// TwinCAT 3 PLC project TPA
// ProgramVersion: 3.1.4023.0
// libraries:
//   Tc2_MC2, * (Beckhoff Automation GmbH)
//   Tc2_Standard, * (Beckhoff Automation GmbH)
//   Tc2_System, * (Beckhoff Automation GmbH)
//   Tc2_Utilities, * (Beckhoff Automation GmbH)
//   Tc3_Module, * (Beckhoff Automation GmbH)
//   VisuSymbols,3.5.10.0,System
// project tree:
//   / GlobalTextList.TcGTLO, PlcTask.TcTTO, Visualization Manager.TcVMO (not stored)
//   GVLs/ GVL.TcGVL
//   POUs/ MAIN.TcPOU, PlixHandler.TcPOU, POU.TcPOU
//   VISUs/ Visualization.TcVIS
// real-time tasks:
//   TASK PlcTask: cycle T#10ms, priority 20, ADS port 350
// motion (NC):
//   TASK NC-Task 1 SAF: cycle T#2ms, priority 4, ADS port 501
//   TASK NC-Task 1 SVB: cycle T#10ms, priority 8, ADS port 511
//   AXIS Axis 1 (id 1)
//     Dynamic: Acceleration=7555.57, Deceleration=7555.57, Jerk=32111.1
//     PositionAreaControl: Range=10
//     TargetPosControl: Range=10, Time=0.05
//     OtherSettings: AllowMotionCmdToSlave=true
//     encoder EncType=4
//       EncPara: ScaleFactorNumerator=0.09, MaxCount=#x0000ffff
//         Inc: RefSoftSyncMask=#x0000ffff
//     drive DrvType=24
//       Analog: VeloReferenz=1800, TorqueSetpointScale=10, ScaleFactorActTorque=0.1
//       TimeComp: TaskDelayCycles=1
//     controller CtrType=1
//       CtrPara: PriorControlFactor=1
//         PosDiffControl: Enable=false
//         Observer: BandWidth=20
// I/O:
//   DEVICE Device 3 (EtherCAT), AmsNetId 192.168.1.97.4.1
//     Box 2 (EasyCAT 32+32 rev 1) [Generic 32+32 bytes rev 1]
//     Term 3 (EK1100) [EK1100 EtherCAT Coupler (2A E-Bus)]
//       Term 4 (EL7041) [EL7041 1Ch. Stepper motor output stage (50V, 5A)]
//       Term 5 (EL9011) [EL9011 End Terminal]
// variable links:
//   NC-Task 1 SAF/Axes/Axis 1 <-> Device 3 (EtherCAT)/Term 3 (EK1100)/Term 4 (EL7041)
//     Drive/Inputs/In/nState1 @bit 3 <-> STM Status/Status/Error
//     Drive/Inputs/In/nState1 @bit 5 <-> STM Status/Status/Moving negative
//     Drive/Inputs/In/nState1 @bit 4 <-> STM Status/Status/Moving positive
//     Drive/Inputs/In/nState1 @bit 1 <-> STM Status/Status/Ready
//     Drive/Inputs/In/nState1 <-> STM Status/Status/Ready to enable
//     Drive/Inputs/In/nState1 @bit 6 <-> STM Status/Status/Torque reduced
//     Drive/Inputs/In/nState1 @bit 2 <-> STM Status/Status/Warning
//     Drive/Inputs/In/nState2 @bit 3 <-> STM Status/Status/Digital input 1
//     Drive/Inputs/In/nState2 @bit 4 <-> STM Status/Status/Digital input 2
//     Drive/Inputs/In/nState2 @bit 5 <-> STM Status/Status/Sync error
//     Drive/Inputs/In/nState2 @bit 7 <-> STM Status/Status/TxPDO Toggle
//     Drive/Inputs/In/nState4 @bit 1 <-> WcState/InputToggle
//     Drive/Inputs/In/nState4 <-> WcState/WcState
//     Drive/Outputs/Out/nCtrl1 <-> STM Control/Control/Enable
//     Drive/Outputs/Out/nCtrl1 @bit 2 <-> STM Control/Control/Reduce torque
//     Drive/Outputs/Out/nCtrl1 @bit 1 <-> STM Control/Control/Reset
//     Drive/Outputs/Out/nDataOut2[0] <-> STM Velocity/Velocity
//     Enc/Inputs/In/nDataIn1[0] <-> ENC Status compact/Counter value
//     Enc/Inputs/In/nDataIn2[0] <-> ENC Status compact/Latch value
//     Enc/Inputs/In/nState1 @bit 4 <-> ENC Status compact/Status/Counter overflow
//     Enc/Inputs/In/nState1 @bit 3 <-> ENC Status compact/Status/Counter underflow
//     Enc/Inputs/In/nState1 @bit 7 <-> ENC Status compact/Status/Extrapolation stall
//     Enc/Inputs/In/nState1 <-> ENC Status compact/Status/Latch C valid
//     Enc/Inputs/In/nState1 @bit 1 <-> ENC Status compact/Status/Latch extern valid
//     Enc/Inputs/In/nState1 @bit 2 <-> ENC Status compact/Status/Set counter done
//     Enc/Inputs/In/nState2 @bit 4 <-> ENC Status compact/Status/Status of extern latch
//     Enc/Inputs/In/nState2 <-> ENC Status compact/Status/Status of input A
//     Enc/Inputs/In/nState2 @bit 1 <-> ENC Status compact/Status/Status of input B
//     Enc/Inputs/In/nState2 @bit 2 <-> ENC Status compact/Status/Status of input C
//     Enc/Inputs/In/nState2 @bit 5 <-> ENC Status compact/Status/Sync error
//     Enc/Inputs/In/nState2 @bit 7 <-> ENC Status compact/Status/TxPDO Toggle
//     Enc/Inputs/In/nState4 @bit 1 <-> WcState/InputToggle
//     Enc/Inputs/In/nState4 <-> WcState/WcState
//     Enc/Outputs/Out/nCtrl1 <-> ENC Control compact/Control/Enable latch C
//     Enc/Outputs/Out/nCtrl1 @bit 3 <-> ENC Control compact/Control/Enable latch extern on negative edge
//     Enc/Outputs/Out/nCtrl1 @bit 1 <-> ENC Control compact/Control/Enable latch extern on positive edge
//     Enc/Outputs/Out/nCtrl1 @bit 2 <-> ENC Control compact/Control/Set counter
//     Enc/Outputs/Out/nDataOut1[0] <-> ENC Control compact/Set counter value
//   TPA/TPA Instance <-> Device 3 (EtherCAT)/Box 2 (EasyCAT 32+32 rev 1)
//     PlcTask Inputs/GVL.Analog1 <-> Inputs/Byte0
//     PlcTask Inputs/GVL.Analog2 <-> Inputs/Byte1
//     PlcTask Inputs/GVL.Analog3 <-> Inputs/Byte2
//     PlcTask Inputs/GVL.Average <-> Inputs/Byte3
//     PlcTask Inputs/GVL.Byte31IN <-> Inputs/Byte31
//     PlcTask Inputs/GVL.Sensors <-> Inputs/Byte12
//     PlcTask Outputs/GVL.ArduinoState <-> Outputs/Byte0
//     PlcTask Outputs/GVL.FanDyno <-> Outputs/Byte1
//     PlcTask Outputs/GVL.OutArduino2 <-> Outputs/Byte2
//     PlcTask Outputs/GVL.OutArduino3 <-> Outputs/Byte3
//     PlcTask Outputs/GVL.WingSpeed <-> Outputs/Byte4
//   TPA/TPA Instance <-> NC-Task 1 SAF/Axes/Axis 1
//     PlcTask Inputs/GVL.StackStepper.NcToPlc <-> Outputs/ToPlc
//     PlcTask Outputs/GVL.StackStepper.PlcToNc <-> Inputs/FromPlc

CONFIGURATION TPA
    RESOURCE PLC ON TwinCAT3
        TASK PlcTask(INTERVAL := T#10ms, PRIORITY := 20);
        PROGRAM MAIN WITH PlcTask : MAIN;
    END_RESOURCE
END_CONFIGURATION

// ---- GVLs/GVL.TcGVL
{attribute 'qualified_only'}
VAR_GLOBAL
	
	//Timing				/////////////////////////////////////////			
	SystemTime							:WORD;
	SystemTimeM							:WORD;
	SystemTimeMs						:WORD;
	ArduinoComsTimer					:TON;
	ArduinoComsTime						:TIME		:=T#20MS;
		
	//Arduino				/////////////////////////////////////////
		//States
	ArduinoState 				AT %Q*	:USINT		:=0;//byte out 0
	FanDyno						AT %Q*	:USINT		:=0;//byte out 1
	OutArduino2					AT %Q*	:BYTE;			//byte out 2
	OutArduino3					AT %Q*	:BYTE;			//byte out 3
	WingSpeed					AT %Q*	:USINT		:=30;//byte out 4
	Idle						:USINT	:= 0;
	
	Byte31IN					AT %I*	:USINT;
	TopEndStop					AT %I*	:BOOL;
	BottomEndStop				AT %I*	:BOOL;
	Analog1   					AT %I*	:USINT;			//byte in 0
	Analog2   					AT %I*	:USINT;			//byte in 1
	Analog3   					AT %I*	:USINT;			//byte in 2
	Average   					AT %I*	:USINT;			//byte in 3
	Sensors						AT %I*	:USINT;			//byte in 12
	Sensors2						AT %I*	:USINT;			//byte in 13
	
		
		//Inputs
	ArduinoBusyBit			:BOOL;
	
		//Outputs
PlixShooter			: BOOL;	//Pin2224V;
StackBlast			: BOOL;	//Pin2324V;
DoubleJets			: BOOL;	//Pin2424V;
CarriageWaitRam		: BOOL;	//Pin2524V;
CarriageRam			: BOOL;	//Pin2624V;
BoxGripper			: BOOL;	//Pin2724V;
BoxGrabber			: BOOL;	//Pin2824V;
FlapFolder1			: BOOL;	//Pin2924V;
FlapFolder2			: BOOL;	//Pin3024V;
BoxCart				: BOOL;	//Pin3124V;
TopClamp			: BOOL;	//Pin3224V;
BottomClamp			: BOOL;	//Pin3324V;
BoxSizeAdjust		: BOOL;	//Pin3424V;
o2					: BOOL;	//Pin3524V;
o3					: BOOL;	//Pin3624V;
o4					: BOOL;	//Pin3724V;
	
	//Stepper				/////////////////////////////////////////
	StackStepper : axis_ref;

	PlixInBox: BOOL;
END_VAR

// ---- POUs/MAIN.TcPOU
PROGRAM MAIN
VAR



	
	//Varibles				/////////////////////////////////////////
	e 						:INT;
	
	TopPickCut				:INT;
	HalfWayCut				:INT;
	TopPickScan				:INT;
	HalfWayDownScan			:INT;
	PlixInBox				:BOOL; //if theres a plix in the box 
	
	
	


	
	//Unsure				/////////////////////////////////////////
	msgCtrlMask     		:DWORD;
    msgFmtStr               :T_MaxString;
    strArg          		:T_MaxString;

	
	//Time					/////////////////////////////////////////
	fbTime					:FB_LocalSystemTime := ( bEnable :=TRUE, dwCycle := 1 );
	StartTime				:REAL;
	GoTime					:REAL;
	
	TotalTime				:REAL;
	
	TimeSeconds				:REAL;
	Delay 					:TON;
	
	PlixHandlerFB : PlixHandler;
END_VAR


//Arduino					/////////////////////////////////////////
	//IO Setup
GVL.OutArduino2.0 := GVL.PlixShooter;		//Pin2224V;
GVL.OutArduino2.1 := GVL.StackBlast;		//Pin2324V;
GVL.OutArduino2.2 := GVL.DoubleJets;		//Pin2424V;
GVL.OutArduino2.3 := GVL.CarriageWaitRam;	//Pin2524V;
GVL.OutArduino2.4 := GVL.CarriageRam;		//Pin2624V;
GVL.OutArduino2.5 := GVL.BoxGripper;		//Pin2724V;
GVL.OutArduino2.6 := GVL.BoxGrabber;		//Pin2824V;
GVL.OutArduino2.7 := GVL.FlapFolder1;		//Pin2924V;
GVL.OutArduino3.7 := GVL.FlapFolder2;		//Pin3024V;
GVL.OutArduino3.6 := GVL.BoxCart;			//Pin3124V;
GVL.OutArduino3.5 := GVL.TopClamp;			//Pin3224V;
GVL.OutArduino3.4 := GVL.BottomClamp;		//Pin3324V;
GVL.OutArduino3.3 := GVL.BoxSizeAdjust;		//Pin3424V;
GVL.OutArduino3.2 := GVL.o2;				//Pin3524V;
GVL.OutArduino3.1 := GVL.o3;				//Pin3624V;
GVL.OutArduino3.0 := GVL.o4;				//Pin3724V;
GVL.ArduinoBusyBit := GVL.Byte31IN.0;
PlixHandlerFB(
	go :=TRUE,
	);
GVL.ArduinoComsTimer(
	IN := GVL.ArduinoState > 0,
	PT := GVL.ArduinoComsTime,);
	
IF GVL.ArduinoComsTimer.Q THEN
	GVL.ArduinoState := GVL.Idle;
END_IF
	//Plix in Box
//IF (NOT Sensor3 AND Sensor2) THEN
//	PlixInBox := TRUE;
//ELSE 
//	PlixInBox := FALSE;
//END_IF


//Time SetUp				/////////////////////////////////////////	
GVL.SystemTime := fbTime.systemTime.wSecond;
GVL.SystemTimeMs := fbTime.systemTime.wMilliseconds;
GVL.SystemTimeM := fbTime.systemTime.wMinute;
TimeSeconds := GVL.SystemTime + (GVL.SystemTimeMs * 0.001) + ( GVL.SystemTimeM * 60 );
fbTime();

END_PROGRAM

// ---- POUs/PlixHandler.TcPOU
FUNCTION_BLOCK PlixHandler
VAR_INPUT
	go :BOOL;

END_VAR
VAR_OUTPUT
	

END_VAR
VAR
	//Arduino				/////////////////////////////////////////
		//States
	Scanner					:USINT		:= 10;
	
		//Varibles
	WingUp					:USINT 		:=220;
	WingFlat				:USINT 		:=180;
	WingHDown				:USINT 		:=155;
	WingDown				:USINT 		:=80;
	WiggleDown				:USINT 		:=155;
	WiggleUP				:USINT 		:=190;
	FanHigh					:USINT 		:=115;
	FanLow					:USINT 		:=95;
	FanOff					:USINT 		:=89;
	FanReverse				:USINT 		:=74;
	WingGo					:USINT		:=20;
	FanGo					:USINT		:=30;

	//Stepper				/////////////////////////////////////////
	HaltStackStepper	: MC_Halt;
	EnableStackStepper	: MC_Power;
	MoveStackAbsolute	: MC_MoveAbsolute;
	ReadStackPosition	: MC_ReadActualPosition;
	SetStackPosition	: MC_SetPosition;
	StopStackStepper	: MC_Stop;
	ResetStackStepper	: MC_Reset;
	
		//Varibles
	StackStepperRun: BOOL;
	StackStepperPosition: LREAL;
	StackStepperVelocity: LREAL;
	StackStepperCurrentPosition: LREAL;
	StackStepperZeroPosition : BOOL;
	StackStepperStop: BOOL;
	StackStepperReset: BOOL;
	StackStepperHalt: BOOL;
	StackStepperHaltDone: BOOL;
	StackStepperAbsoluteDone: BOOL;
	StackStepperEnable: BOOL;
	
	Byte31IN: BYTE;
	StackSensor1: BOOL;
	Sensors: BYTE;
	StackSensor2: BOOL;
	StackSensor3: BOOL;
	Sensor4: BOOL;
	Sensor5: BOOL;
	PlixHandlerState: INT;
	BottomEndStop: BOOL;
	Boot: BOOL := TRUE;
	Calibrate 				:BOOL;
	NextState: INT;
	Single					:BOOL;
	Double					:BOOL;
	Zero					:BOOL;
	Start					:BOOL;
	//Stats					/////////////////////////////////////////
	Singles					:INT;
	Doubles					:INT;
	Zeros					:INT;
	Total					:INT;
	Wiggle					:INT;
	Count 					:INT		:= 0;
	Delay 					:TON;
	CycleTime				:REAL;
	EndTime					:REAL;
	AverageTime				:REAL;
	DoubleLoop: INT;
	Blast: BOOL;
	Cali: INT	 :=0;
	Velocity 				:LREAL :=1000;
	ErrorID1		        : UDINT;
	
END_VAR
VAR PERSISTENT				/////////////////////////////////////////
	
	//CutPoints				/////////////////////////////////////////
	PlixNumberScan			:INT;
	PlixNumberScanLeft		:INT;
	PlixNumberScanRight		:INT;
	NormalTopCut			:UINT;
	NormalBottomCut			:UINT;
	TopCut					:UINT;
	BottomCut				:UINT;
	DoubleTopCut			:UINT;
	DoubleBottomCut			:UINT;
	TopCutLeft				:INT;
	BottomCutLeft			:INT;
	TopCutRight				:INT;
	BottomCutRight			:INT;
	
	
	//Time					/////////////////////////////////////////

END_VAR

MoveStackAbsolute(
	Axis:= GVL.StackStepper, 
	Execute:= StackStepperRun, 
	Position:= StackStepperPosition, 
	Velocity:= StackStepperVelocity, 
	Acceleration:= 7555.57, 
	Deceleration:= 7555.57, 
	Jerk:= 32111.1,
	Done=> StackStepperAbsoluteDone, );
	
HaltStackStepper(
	Axis:= GVL.StackStepper, 
	Execute:= StackStepperHalt, 
	Deceleration:= 7555.57,  
	Done=> StackStepperHaltDone,
	ErrorID=> ErrorID1, );
	
EnableStackStepper(
	Axis:= GVL.StackStepper, 
	Enable:= StackStepperEnable, 
	Enable_Positive:= StackStepperEnable, 
	Enable_Negative:= StackStepperEnable, );

ReadStackPosition(
	Axis:= GVL.StackStepper, 
	Enable:= StackStepperEnable, 
	Position=> StackStepperCurrentPosition);	

SetStackPosition(
	Axis:= GVL.StackStepper, 
	Execute:= StackStepperZeroPosition, 
	Position:= 0, 
	Mode:= FALSE, 
	Options:= , 
	 );
	
StopStackStepper(
	Axis:= GVL.StackStepper, 
	Execute:= StackStepperStop, 
	Deceleration:= , 
	Jerk:= , 
	Options:= , 
	Done=> , 
	Busy=> , 
	Active=> , 
	CommandAborted=> , 
	Error=> , 
	ErrorID=> );
	
ResetStackStepper(
	Axis:= GVL.StackStepper, 
	Execute:= StackStepperReset, 
	Done=> , 
	Busy=> , 
	Error=> , 
	ErrorID=> );
	
	
	
	
	//Coms

IF go THEN
	StackStepperEnable := TRUE;
END_IF
StackSensor2 := GVL.Sensors.1;
BottomEndStop :=GVL.Sensors.2;
//StackStepperZeroPosition := TRUE;//sometimes after many restarts the position can be massive and cause problems 


CASE PlixHandlerState OF
	
	1:
		StackStepperZeroPosition := FALSE;
		StackStepperRun := FALSE;
		StackStepperHalt :=TRUE;
		IF StackStepperHaltDone THEN 
				PlixHandlerState :=NextState;
				StackStepperHalt :=FALSE;
		END_IF
		
	
	10:	
		IF Boot THEN
			StackStepperZeroPosition := TRUE;
			PlixHandlerState := 11;
		ELSE
			PlixHandlerState := 100;
		END_IF
		
	11://home bottom sensor
		StackStepperZeroPosition := FALSE;
		IF  BottomEndStop THEN//if not blocked drive down till blocked
			StackStepperPosition := -5000;
			StackStepperVelocity := 100;
			StackStepperRun := TRUE;
		ELSE 
			NextState :=20;
			PlixHandlerState :=1;
				
		END_IF
		
	20:
		IF  NOT BottomEndStop THEN//drive up till unblocked
			StackStepperPosition := 8000;
			StackStepperVelocity := 100;
			StackStepperRun := TRUE;
		ELSE 
			NextState :=30;
			PlixHandlerState :=1;	
		END_IF	
		
	30:
		Boot := FALSE;
		StackStepperZeroPosition := TRUE;//set position to zero just above endstop
		//StackStepperZeroPosition := FALSE;
		PlixHandlerState :=100;
	
	100:// home stack top
		StackStepperZeroPosition := FALSE;
		IF NOT StackSensor2 THEN//AND NOT StackSensor2 AND NOT StackSensor3 THEN
			StackStepperPosition := 200;
			StackStepperVelocity := Velocity;//make sure to change the amount of steps to plix pick up
			StackStepperRun := TRUE;
		ELSE 
			NextState :=200;
			PlixHandlerState :=1;
			
		END_IF
	200:
		StackStepperHalt :=FALSE;
		IF StackSensor2 THEN//AND  StackSensor2 AND  StackSensor3 THEN
			StackStepperPosition := 10000;
			StackStepperVelocity := Velocity;//make sure to change the amount of steps to plix pick up
			StackStepperRun := TRUE;
		ELSE 
			NextState :=300;
			PlixHandlerState :=1;
				
		END_IF
	300://fan on
		IF GVL.ArduinoBusyBit THEN//if  arduino is free then ask to change state
			GVL.FanDyno := FanHigh;
			GVL.ArduinoState := FanGo;
			PlixHandlerState :=400;
		END_IF
		
	400://up to head
		IF Blast THEN 
			GVL.StackBlast := TRUE;
		END_IF
		Blast := FALSE;
		StackStepperHalt :=FALSE;
		StackStepperPosition := StackStepperCurrentPosition + 50;
		StackStepperVelocity := Velocity;
		StackStepperRun := TRUE;
		PlixHandlerState :=500;
		
	500://down
		
		StackStepperRun := FALSE;
		IF StackStepperAbsoluteDone THEN
			GVL.StackBlast := FALSE;
		/////
			
			StackStepperPosition := StackStepperCurrentPosition - 400;
			StackStepperVelocity := Velocity;//make sure to change the amount of steps to plix pick up
			StackStepperRun := TRUE;
			StackStepperAbsoluteDone := FALSE;
			PlixHandlerState :=550;
			
		END_IF
		
	550:
		StackStepperRun := FALSE;
		IF StackStepperAbsoluteDone THEN
			NextState :=575;
			PlixHandlerState :=1;
				
		END_IF
		
	575:
		IF Calibrate THEN
			PlixHandlerState :=580;
		ELSE
			PlixHandlerState :=600;
		END_IF
		
	580:
		Delay(IN:=TRUE, PT:=T#1000MS);
      	IF Delay.Q THEN
        	Delay(IN:=FALSE);
			
			PlixHandlerState :=600;
		END_IF
	600://scan
		
		IF GVL.ArduinoBusyBit THEN//if arduino is free then ask to change state
			GVL.ArduinoState := Scanner;
			PlixHandlerState :=700;
		END_IF
	
	700:
		IF GVL.ArduinoBusyBit THEN//if arduino is free then ask to change state
			PlixHandlerState :=800;
		END_IF
	800://still hasnt written the new scan to beckhoff so we need to wait a little for it to loop on the arduino
	Delay(IN:=TRUE, PT:=T#500MS);
      	IF Delay.Q THEN
        	Delay(IN:=FALSE);
			
			PlixHandlerState :=900;
		END_IF
	900:
		IF NOT Calibrate THEN
			IF DoubleLoop > 0 THEN
				TopCut := DoubleTopCut;
				BottomCut := DoubleBottomCut;
				PlixHandlerState :=1000;
			ELSE
				TopCut := NormalTopCut;
				BottomCut := NormalBottomCut;
				PlixHandlerState :=1000;
			END_IF
		ELSE 
			PlixHandlerState :=1000;
		END_IF
	1000://decision
		IF GVL.Average > TopCut THEN
			Zero := TRUE;
			Blast := TRUE;
			PlixHandlerState :=2500;
		
		ELSIF  GVL.Average <= TopCut AND GVL.Average > BottomCut THEN
			Single := TRUE;
			PlixHandlerState :=2000;
			
		ELSIF GVL.Average <= BottomCut THEN
			
			Blast := TRUE;
			DoubleLoop := DoubleLoop +1;
			WiggleDown := WiggleDown - 25;
			WiggleUP := WiggleUP + 10;
			PlixHandlerState :=1025;
			
		END_IF
		IF Calibrate THEN
			IF Cali = 0 THEN
				Single := TRUE;
				NormalTopCut := GVL.Average + 100;
				NormalBottomCut := GVL.Average - 10;
				PlixHandlerState :=1025;
			ELSIF Cali = 1 THEN
				DoubleTopCut := GVL.Average + 100;
				DoubleBottomCut := GVL.Average - 20;
				PlixHandlerState :=2500;
			END_IF	
		END_IF
	//zero
		//blast stack
		//repick
	//double
		//wiggle
		//blast
		//rescan
	1025:
		IF DoubleLoop <= 1 THEN
			StackStepperPosition := StackStepperCurrentPosition - 150;
			StackStepperVelocity := Velocity;//make sure to change the amount of steps to plix pick up
			StackStepperRun := TRUE;
			PlixHandlerState :=1030;
		ELSE
			PlixHandlerState :=1050;
		END_IF
	1030:
		StackStepperRun := FALSE;
		
		IF StackStepperAbsoluteDone THEN
			Cali := 1;
			PlixHandlerState :=575;
		END_IF
	1050:
		
			IF DoubleLoop > 5 THEN
				Total := Total + 2;
				Double := TRUE;
				
				PlixHandlerState :=2000;
			ELSE
				PlixHandlerState :=1100;
			END_IF
		
	1100:
		Wiggle := Wiggle +1;
		IF GVL.ArduinoBusyBit THEN//if arduino is free then ask to change state
			GVL.WingSpeed := 60;
			GVL.FanDyno := WiggleDown;
			GVL.ArduinoState := WingGo;
			Delay(IN:=TRUE, PT:=T#500MS);
			IF Delay.Q THEN
				Delay(IN:=FALSE);
				GVL.DoubleJets := TRUE;
				//GVL.LeftAirJet := TRUE;
				PlixHandlerState := 1200; 
			END_IF
		END_IF
	1200:
		IF GVL.ArduinoBusyBit THEN//if arduino is free then ask to change state
			GVL.WingSpeed := 20;
			GVL.FanDyno := WiggleUP;
			GVL.ArduinoState := WingGo;
			Delay(IN:=TRUE, PT:=T#500MS);
			IF Delay.Q THEN
				Delay(IN:=FALSE);
				GVL.DoubleJets := FALSE;
				//GVL.RightAirJet := FALSE;
				PlixHandlerState := 1300;
			END_IF
		END_IF
	1300:
		IF GVL.ArduinoBusyBit THEN
			GVL.WingSpeed := 60;
			GVL.FanDyno :=WingFlat;
			GVL.ArduinoState := WingGo;
			
			Delay(IN:=TRUE, PT:=T#500MS);
			IF Delay.Q THEN
				Delay(IN:=FALSE);
				PlixHandlerState := 600;
			END_IF
		END_IF
	
	//////////////////////////////////////////////////
		
	2000:
		IF GVL.ArduinoBusyBit THEN
			GVL.FanDyno := 74;
			GVL.ArduinoState := FanGo;
			PlixHandlerState:=2200;
		END_IF
	2200:
			//GVL.FanDyno := 74;
			//GVL.ArduinoState := FanGo;
		Delay(IN:=TRUE, PT:=T#300MS);
		IF Delay.Q THEN
        	Delay(IN:=FALSE);
        	PlixHandlerState := 2300;
    	END_IF
	2300:
		IF GVL.ArduinoBusyBit THEN
			GVL.PlixShooter :=TRUE;
			PlixHandlerState := 2400;
		END_IF
	2400:
		Delay(IN:=TRUE, PT:=T#300MS);
		IF Delay.Q THEN
        	Delay(IN:=FALSE);
        	PlixHandlerState := 2500;
    	END_IF
	2500:
		IF GVL.ArduinoBusyBit THEN
			GVL.FanDyno := 89;
			GVL.ArduinoState := FanGo;
			PlixHandlerState := 2600;
		END_IF
	2600:
		Delay(IN:=TRUE, PT:=T#100MS);
		IF Delay.Q THEN
        	Delay(IN:=FALSE);
			GVL.PlixShooter :=FALSE;
        	PlixHandlerState := 2800;
    	END_IF
	2800:
	//finishing up stats ant time and stuff
		PlixHandlerState :=100;
		DoubleLoop := 0;
		WiggleDown := 155;
		WiggleUP := 190;
		IF Single THEN
			Singles := Singles +1;
			Total := Total + 1;
		END_IF
		IF Double THEN
			Doubles := Doubles +1;
		END_IF
		Single := FALSE;
		Double := FALSE;
		EndTime := MAIN.TimeSeconds;	
		IF Singles > 1 THEN
			AverageTime := (EndTime - MAIN.GoTime)/Singles;
		END_IF
		
		CycleTime := EndTime - MAIN.StartTime;
		IF Calibrate THEN
			Singles := Singles -1;
			Blast := FALSE;
			Cali := 0;
			//TopCutLeft := GVL.AverageLeft - 40;
			//BottomCutLeft := AverageLeft - 66;
			//TopCutRight := AverageRight + 10;
			//BottomCutRight := AverageRight - 50;
			PlixHandlerState :=0;
			Calibrate := FALSE;
		END_IF
		
	
END_CASE

END_FUNCTION_BLOCK

// ---- POUs/POU.TcPOU
FUNCTION_BLOCK POU
VAR_INPUT
END_VAR
VAR_OUTPUT
END_VAR
VAR
	//STATES				/////////////////////////////////////////
		BoxRemoved						: BOOL;
		PlixRequest						: BOOL;
		BoxGrabbed						: BOOL;
		BoxRemoverState					: INT;
		BoxReady						: BOOL;
		BoxDropRequest					: BOOL;
		BoxDelivered					: BOOL;
		BoxCartHome						: BOOL;
		BoxLoaderState					: INT;
		FlapFolderState					: INT;
		BoxGraberState					: INT;
		BoxDropped 						: BOOL;
		BoxRemover						: INT :=0;
		BoxStackNeeded					: BOOL;
		BoxRefillState					: INT;
		
	//ARDUINO				/////////////////////////////////////////
	
		//INPUTS
	
			PlixSensor1					: BOOL; //sensor
			PlixSensor2					: BOOL; //sensor
			MainStackFull				: BOOL; //sensor
			SecondaryStackFull			: BOOL; //sensor
			LastBoxGone					: BOOL; //sensor
			BoxGrabberUp				: BOOL;//sensor
			BoxGrabberDown				: BOOL;//sensor
			FlapFolder1Up				: BOOL;//Sensor
			FlapFolder1Down				: BOOL;//Sensor
			FlapFolder2Up				: BOOL;//Sensor
			FlapFolder2Down				: BOOL;//Sensor
			CarriageAtPickUp			: BOOL; //sensor
			CarriageAtDrop 				: BOOL;//sensor
					
		//OUTPUTS
			CarriageWaitRam				: BOOL;
			CarriageRam					: BOOL;
			BoxGripper					: BOOL;
			BoxGrabber					: BOOL;
			FlapFolder1					: BOOL;
			FlapFolder2					: BOOL;
			BoxCart						: BOOL;
			TopClamp					: BOOL;
			BottomClamp					: BOOL;
			
			
	//TIME					/////////////////////////////////////////
		BoxCartTimer					: TON;
		BoxCartTime						: TIME := T#2000MS;
		FlapResetTimer					: TON;
		FlapResetTime					: TIME := T#500MS;
		BoxDropTimer					: TON;
		BoxDropTime						: TIME := T#500MS;
		PlixFlightTimer 				: TON;
		PlixFlightTime 					: TIME := T#500MS;
	
	
		StackReadyToDrop: BOOL;
END_VAR

//need the code to decide when the boxes get dropped onto the gripper for a box refil



//need timer for how long boxes have been on cart, make sure theyre stable(maybe a button to say ready
BoxCartTimer(
	IN := BoxCart = TRUE,
	PT := BoxCartTime,);

FlapResetTimer(//dont need this as we have the sensors 
	IN := FlapFolder2 = FALSE,
	PT := FlapResetTime,);
	
BoxDropTimer(//boxes dropped onto the graber before its gripped and pulled off
	IN := BottomClamp = FALSE,
	PT := BoxDropTime,);
	
PlixFlightTimer(//time from the head shooting the plix to it landing in a box
	IN := PlixRequest = FALSE,
	PT := PlixFlightTime,);

	
PlixSensor1		 	:= GVL.Sensors.3;
PlixSensor2 		:= GVL.Sensors.4;
MainStackFull 		:= GVL.Sensors.5;
SecondaryStackFull 	:= GVL.Sensors.6;
LastBoxGone 		:= GVL.Sensors.7;
BoxGrabberUp 		:= GVL.Sensors2.0;
BoxGrabberDown		:= GVL.Sensors2.1;
FlapFolder1Up		:= GVL.Sensors2.2;
FlapFolder1Down		:= GVL.Sensors2.3;
FlapFolder2Up 		:= GVL.Sensors2.4;
FlapFolder2Down 	:= GVL.Sensors2.5;
CarriageAtPickUp 	:= GVL.Sensors2.6;
CarriageAtDrop 		:= GVL.Sensors2.7;
	
	
	
CASE BoxLoaderState OF
	100: //idle state moves the box cart to the loading position and waits for boxes to be put on
		BoxCart := FALSE;
		BoxCartHome := TRUE;//so we know were at the home end of the rams travel
		BoxLoaderState := 200;
		
	200:// if we have boxes in the cart and there are no boxes in the machine and clamp is open we move the stack over
		IF MainStackFull AND NOT SecondaryStackFull AND BoxCartHome AND NOT TopClamp  THEN
			BoxCart := TRUE;
			BoxCartHome := FALSE;
			BoxCartTimer := TRUE;
			BoxLoaderState := 210;
			
		END_IF//move boxes over if no boxes left and stack ready to load.
	210:
		IF BoxCartTimer.Q AND SecondaryStackFull THEN//after timer and if stack is on the cart we clamp it in place.
			TopClamp:=TRUE;
			BoxLoaderState :=300;
		END_IF
		
	300:
		IF TopClamp AND SecondaryStackFull THEN//once clamped we remove the cart ready to drop stack 
			BoxCart := FALSE;
			//TopClamp := TRUE;
			BoxCartHome := TRUE;
			BoxCartTimer := TRUE;
			StackReadyToDrop := TRUE;
			BoxLoaderState := 400;
		END_IF
	400:	
		IF NOT StackReadyToDrop THEN
			BoxLoaderState := 100;
		END_IF
		
END_CASE
CASE FlapFolderState OF
	100:
		FlapFolder1 := FALSE;
		FlapFolder2 := FALSE;
		BoxGripper := FALSE;
		FlapResetTimer := TRUE;
		FlapFolderState := 200;
		
	200:
		IF FlapFolder1Up AND FlapFolder2Up THEN
			BoxGrabber :=TRUE;
			BoxGripper :=FALSE;
			FlapFolderState := 300;
		END_IF
	210: 
		IF NOT MainStackFull THEN //if theres no boxes we say no boxes and wait for that to be sorted
			BoxStackNeeded := TRUE;
			BottomClamp := FALSE;//drops the boxes on to the gripper
			FlapFolderState := 300;
		ELSE
			FlapFolderState := 310;//if we have boxes carry on
		END_IF
	300: 
		IF NOT BoxStackNeeded THEN
			FlapFolderState := 310;//once boxes are loaded we carry on
		END_IF
	310:
		IF BoxGrabberUp THEN
			BottomClamp := FALSE;//drops the boxes on to the gripper
			FlapFolderState := 400;
		END_IF
		
		
		
	400:
		IF BoxDropTimer.Q THEN//after a small timer for drop the stack is gripped again
			BottomClamp :=TRUE;//after timer finnished 
			BoxGripper :=TRUE;
			FlapFolderState := 500;
		END_IF
		
	500:	//may need a timer here 
		BoxGrabber := FALSE;//box in the grabber is pulled off bottom of the stack
		FlapFolderState := 600;
		
	600:
		IF BoxGrabberDown THEN
			FlapFolder1 := TRUE;
			PlixRequest := TRUE;//must be set false in plix handler aftr shot
			FlapFolderState := 610;
		END_IF
		
	610:
		IF FlapFolder1Down THEN
			FlapFolderState :=710;
		END_IF
		
	710:
		IF NOT PlixRequest	THEN
			//plix has been shot by plix head 
			FlapFolderState := 720;
		END_IF
		
	720:
		//timer to wait a sec for plix to fly
		IF PlixFlightTimer.Q THEN
			FlapFolderState := 730;
		END_IF
	730:
		IF NOT PlixSensor1 AND PlixSensor2 THEN
			FlapFolder2 := TRUE;
			FlapFolderState := 800;
		END_IF
	800: 
		IF FlapFolder2Down THEN
			BoxReady := TRUE;
			FlapFolderState := 810;
		END_IF
		
	
	810:
		IF BoxGrabbed THEN
			BoxGripper := FALSE;
			FlapFolderState := 820;
		END_IF
	820:
		IF BoxRemoved THEN 
			FlapFolderState := 100;
		END_IF
END_CASE




CASE BoxRemoverState OF
	100:
		IF CarriageAtPickUp AND NOT BoxDropped THEN //if  carrige at pick up when turned on 
			CarriageRam :=TRUE; //start it going to drop end
			BoxRemoverState := 200;
		END_IF
		
	200:
		IF NOT CarriageAtPickUp THEN //soon as not at pick up 
			CarriageWaitRam := TRUE;//turn on wait ram 
			CarriageRam :=FALSE;// start carridge coming back to pick up
			BoxRemoverState := 300;
		END_IF
		
	300:
		IF CarriageAtPickUp AND BoxReady THEN
			CarriageWaitRam :=FALSE;
			BoxRemoverState := 400;
		END_IF
	400: 
		BoxReady := FALSE;
		BoxGrabbed := TRUE;
		BoxRemoverState := 500;
	500:
		IF NOT BoxGripper THEN
			CarriageRam := TRUE;
			BoxRemoverState := 600;
		END_IF
		
	600:
		IF CarriageAtDrop AND BoxDropRequest THEN
			CarriageWaitRam := TRUE;
			BoxGrabbed := FALSE;
			BoxRemoverState := 700;
		END_IF
	700: 
		IF BoxDropped THEN
			BoxDelivered :=TRUE;
			BoxRemoverState := 200;
		END_IF
END_CASE

CASE BoxRefillState OF
	100:
		IF BoxStackNeeded THEN
			BoxRefillState := 200;
		END_IF
		
	200:
		IF StackReadyToDrop THEN
			BoxRefillState := 300;
		END_IF
	300:
		StackReadyToDrop := FALSE;
		BoxStackNeeded := FALSE;
		TopClamp:= FALSE;
		BoxRefillState := 100;
END_CASE

END_FUNCTION_BLOCK

// ---- GlobalTextList.TcGTLO
TEXTLIST GlobalTextList
  481 = '%d'
  432 = '%f'
  79 = 'Average'
  745 = 'Blast Air'
  930 = 'box clamp'
  769 = 'Box Grabbed'
  334 = 'BoxD'
  196 = 'BoxReady'
  656 = 'Calibrate'
  311 = 'Cycle'
  625 = 'doubles'
  953 = 'Down'
  71 = 'down'
  509 = 'dpubles'
  890 = 'Dry Run'
  17 = 'Encoder zero'
  197 = 'Fan'
  680 = 'flat'
  214 = 'GO'
  969 = 'Half Down'
  638 = 'High'
  143 = 'Hold'
  690 = 'ignore conveyer'
  576 = 'ignore plix'
  589 = 'ignore stack'
  189 = 'Left Air'
  752 = 'Left Wing'
  971 = 'Mid'
  628 = 'Motor reset'
  61 = 'Motor Reset'
  454 = 'Off'
  750 = 'Reverse'
  187 = 'Right Air'
  681 = 'Right Wing'
  757 = 'Scan'
  942 = 'Shoot Air'
  150 = 'Stop'
  375 = 'up'
  646 = 'WINGS'
  357 = 'Zero stats'
END_TEXTLIST

// ---- VISUs/Visualization.TcVIS
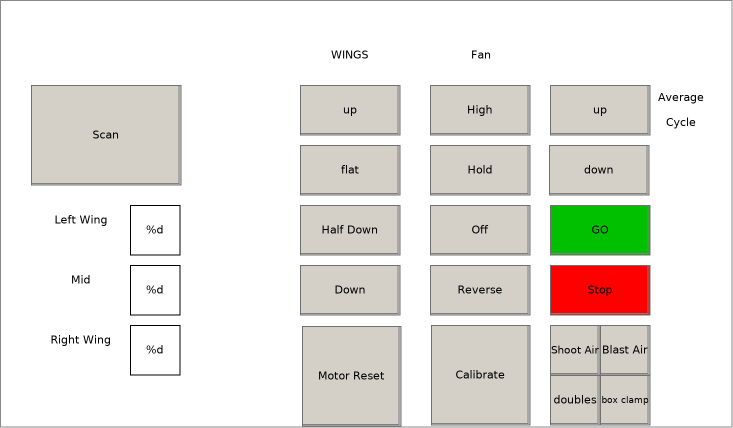
VISUALIZATION Visualization  // 733x428
    Button (31,85 150x100), "Scan"
        OnMouseDown: execute { GVL.ArduinoState := MAIN.PlixHandlerFB.Scanner; }
    Button (300,85 100x50), "up"
        OnMouseDown: execute { GVL.FanDyno := MAIN.PlixHandlerFB.WingUp; GVL.ArduinoState := MAIN.PlixHandlerFB.WingGo; }
    Button (300,145 100x50), "flat"
        OnMouseDown: execute { GVL.FanDyno := MAIN.PlixHandlerFB.WingFlat GVL.ArduinoState :=MAIN.PlixHandlerFB.WingGo }
    Button (300,265 100x50), "Down"
        OnMouseDown: execute { GVL.FanDyno :=MAIN.PlixHandlerFB.WingDown GVL.ArduinoState := MAIN.PlixHandlerFB.WingGo }
    Button (300,205 100x50), "Half Down"
        OnMouseDown: execute { GVL.FanDyno :=MAIN.PlixHandlerFB.WingHDown GVL.ArduinoState := MAIN.PlixHandlerFB.WingGo }
    Label (300,30 100x50), "WINGS"
    Button (430,85 100x50), "High"
        OnMouseDown: execute { GVL.FanDyno := MAIN.PlixHandlerFB.FanHigh; GVL.ArduinoState := MAIN.PlixHandlerFB.FanGo; }
    Button (430,205 100x50), "Off"
        OnMouseDown: execute { GVL.FanDyno :=MAIN.PlixHandlerFB.FanOff GVL.ArduinoState := MAIN.PlixHandlerFB.FanGo }
    Button (430,145 100x50), "Hold"
        OnMouseDown: execute { GVL.FanDyno :=MAIN.PlixHandlerFB.FanLow GVL.ArduinoState := MAIN.PlixHandlerFB.FanGo }
    Label (431,30 100x50), "Fan"
    Button (430,265 100x50), "Reverse"
        OnMouseDown: execute { GVL.FanDyno :=MAIN.PlixHandlerFB.FanReverse GVL.ArduinoState := MAIN.PlixHandlerFB.FanGo }
    Label (631,85 100x25), "Average"
    Label (631,110 100x25), "Cycle"
    Label (31,195 100x50), "Left Wing"
    Label (31,255 100x50), "Mid"
    Label (31,315 100x50), "Right Wing"
    Rectangle (130,205 50x50), "%d"
    Rectangle (130,265 50x50), "%d", text variable: GVL.Average
    Rectangle (130,325 50x50), "%d"
    Button (550,205 100x50), "GO"
        OnMouseUp: execute {
            MAIN.PlixHandlerFB.PlixHandlerState := 10;
            MAIN.GoTime := MAIN.TimeSeconds;
            MAIN.PlixHandlerFB.StackStepperHalt :=FALSE;
            MAIN.POUFB.BoxLoaderState :=100;
            MAIN.POUFB.FlapFolderState :=100;
            MAIN.POUFB.BoxRemoverState :=100;
        }
    Button (550,265 100x50), "Stop"
        OnMouseDown: execute {
            MAIN.PlixHandlerFB.PlixHandlerState := 0;
            GVL.ArduinoState := 0;
            MAIN.PlixHandlerFB.StackStepperStop := TRUE;
            MAIN.PlixHandlerFB.StackStepperRun := FALSE;
            GVL.DoublesJets := FALSE;
            GVL.StackBlast := FALSE;
            GVL.PlixShooter := FALSE;
            MAIN.POUFB.BoxLoaderState :=0;
            MAIN.POUFB.FlapFolderState :=0;
            MAIN.POUFB.BoxRemoverState :=0;
            MAIN.TotalTime := MAIN.TimeSeconds;
        }
        OnMouseUp: execute { MAIN.PlixHandlerFB.StackStepperHalt :=FALSE; MAIN.PlixHandlerFB.Start :=TRUE; }
    Button (550,325 50x50), "Shoot Air"
        OnMouseDown: execute { GVL.PlixShooter := TRUE; }
        OnMouseUp: execute { GVL.PlixShooter := FALSE; }
    Button (600,325 50x50), "Blast Air"
        OnMouseDown: execute { GVL.StackBlast := TRUE; }
        OnMouseUp: execute { GVL.StackBlast := FALSE; }
    Button (550,85 100x50), "up"
    Button (549,145 100x50), "down"
    Button (550,375 50x50), "doubles"
        OnMouseDown: execute { GVL.DoublesJets := TRUE; }
        OnMouseUp: execute { GVL.DoublesJets := FALSE; }
    Button (600,375 50x50), "box clamp"
        OnMouseDown: execute { GVL.BottomClamp := TRUE; }
        OnMouseUp: execute { GVL.BottomClamp := FALSE; }
    Button (431,325 99x100), "Calibrate"
        OnMouseUp: execute { MAIN.PlixHandlerFB.Calibrate := TRUE; MAIN.PlixHandlerFB.PlixHandlerState := 10; }
    Button (302,326 99x100), "Motor Reset"
        OnMouseUp: execute { MAIN.PlixHandlerFB.StackStepperReset := FALSE; }
        OnMouseDown: execute { MAIN.PlixHandlerFB.StackStepperReset := TRUE; MAIN.PlixHandlerFB.StackStepperStop := FALSE; }
END_VISUALIZATION
